Fanuc KAREL source: kt00108.KL

-- PROVISIONAL review KL for V770-1; original PC SHA256 206a804439e01b54af19e798b68288141b8f1bbeb3a5b76d2168c1fbd20f30a5
-- Incomplete behavior may be omitted. Consult companion uncertainty JSON. Do not deploy.
PROGRAM KT00108
%NOLOCKGROUP
VAR
  R1 : REAL
  R2 : REAL
  OUT : REAL
BEGIN
  -- UNRESOLVED_PC offsets 5-16; opcodes 2E,23
  -- UNRESOLVED_PC offsets 21-32; opcodes 2E,23
  -- UNRESOLVED_PC offsets 37-48; opcodes 2E,23
  -- UNRESOLVED_PC offsets 53-64; opcodes 2E,23
  -- UNRESOLVED_PC offsets 69-88; opcodes 21,21,6C,23
  -- UNRESOLVED_PC offsets 93-97; opcodes 7F
END KT00108
